(* Logix 5000 project; controller cal1632 1756-L62 rev 16.20; software revision 16.05; part 7 of 57 *)
(* tags used below, declared in another part *)
   FAULT : BOOL;
   p01_ai_prs : REAL;
   p01_ai_tc : REAL;
   p01_dint_to_hmi : DINT[16];
   p01_int_from_oxidizer : INT[10];
   p01_int_to_oxidizer : INT;
   p01_recipe_active : recipe;
   p01r03_oxidizer_prs : SYS_SCP;
   p01r03_prs_input_max : REAL;
   p01r03_prs_input_min : REAL;
   p01r03_prs_output_max : REAL;
   p01r03_prs_output_min : REAL;
   p01r09_pb_global_reset : BOOL;
   p01r14 : routine;
   p01r14_msg_read : MESSAGE;
   p01r14_msg_read_retry_timer : TIMER;
   p01r14_msg_read_timer : TIMER;
   p01r14_msg_write : MESSAGE;
   p01r14_msg_write_retry_timer : TIMER;
   p01r14_msg_write_timer : TIMER;
   p01r14_oxidizer_heart_beat_off : TIMER;
   p01r14_oxidizer_heart_beat_ok : BOOL;
   p01r14_oxidizer_heart_beat_on : TIMER;
   p01r14_oxidizer_mass_flow : REAL;
   p01r14_timer_fault : TIMER[10];
   p01r14_timer_warning : TIMER[5];
   p02_dint_from_hmi : hmi_dint;
   p02_dint_to_hmi : hmi_dint;
   p02_recipe_from_hmi : recipe;
   p02_recipe_to_hmi : recipe;
   p02r01 : routine;
   p02r02 : routine;
   p02r02_timer_fault : TIMER[4];
   p02r02_timer_logout : TIMER;
   p02r02_timer_warning : TIMER[4];
   p02r03 : routine;
   p02r03_timer_fault : TIMER[4];
   p02r03_timer_warning : TIMER[4];
   p02r04 : routine;
   p02r04_timer_fault : TIMER[4];
   p02r04_timer_warning : TIMER[4];
   p02r05 : routine;
   p02r05_timer_fault : TIMER[4];
   p02r05_timer_warning : TIMER[4];
   p02r07 : routine;
   p11_dint_to_hmi : DINT[16];
   p11r02_shutdown_temp : BOOL;
   p11r20_state : DINT;
   p11r30_request_heat : BOOL;
   p12_dint_to_hmi : DINT[16];
   p12r02_shutdown_temp : BOOL;
   p12r20_state : DINT;
   p12r30_request_heat : BOOL;
   p13_dint_to_hmi : DINT[16];
   p13r02_shutdown_temp : BOOL;
   p13r20_state : DINT;
   p13r30_request_cool : BOOL;
   p19_dint_to_hmi : DINT[16];
   p20_dint_to_hmi : DINT[16];
   p21_dint_to_hmi : DINT[16];
   p22_dint_to_hmi : DINT[16];
   p23_dint_to_hmi : DINT[32];
   p24_dint_to_hmi : DINT[16];
   p25_dint_to_hmi : DINT[16];
   p26_dint_to_hmi : DINT[16];
   p27_dint_to_hmi : DINT[16];
   p28_dint_to_hmi : DINT[16];
   p29_dint_to_hmi : DINT[16];
   p30_dint_to_hmi : DINT[16];
(* P01_System, continued *)

ROUTINE R14_Oxidizer   (* ladder *)
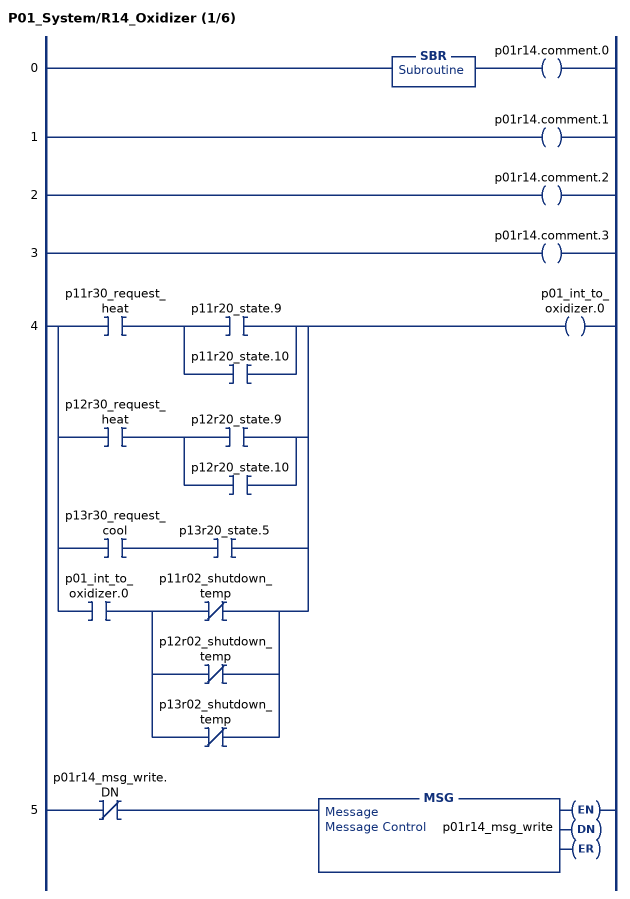
   0: SBR()OTE(p01r14.comment.0);
   1: OTE(p01r14.comment.1);
   2: OTE(p01r14.comment.2);
   3: OTE(p01r14.comment.3);
   4: [XIC(p11r30_request_heat) [XIC(p11r20_state.9) ,XIC(p11r20_state.10) ] ,XIC(p12r30_request_heat) [XIC(p12r20_state.9) ,XIC(p12r20_state.10) ] ,XIC(p13r30_request_cool) XIC(p13r20_state.5) ,XIC(p01_int_to_oxidizer.0) [XIO(p11r02_shutdown_temp) ,XIO(p12r02_shutdown_temp) ,XIO(p13r02_shutdown_temp) ] ]OTE(p01_int_to_oxidizer.0);
   5: XIO(p01r14_msg_write.DN)MSG(p01r14_msg_write);
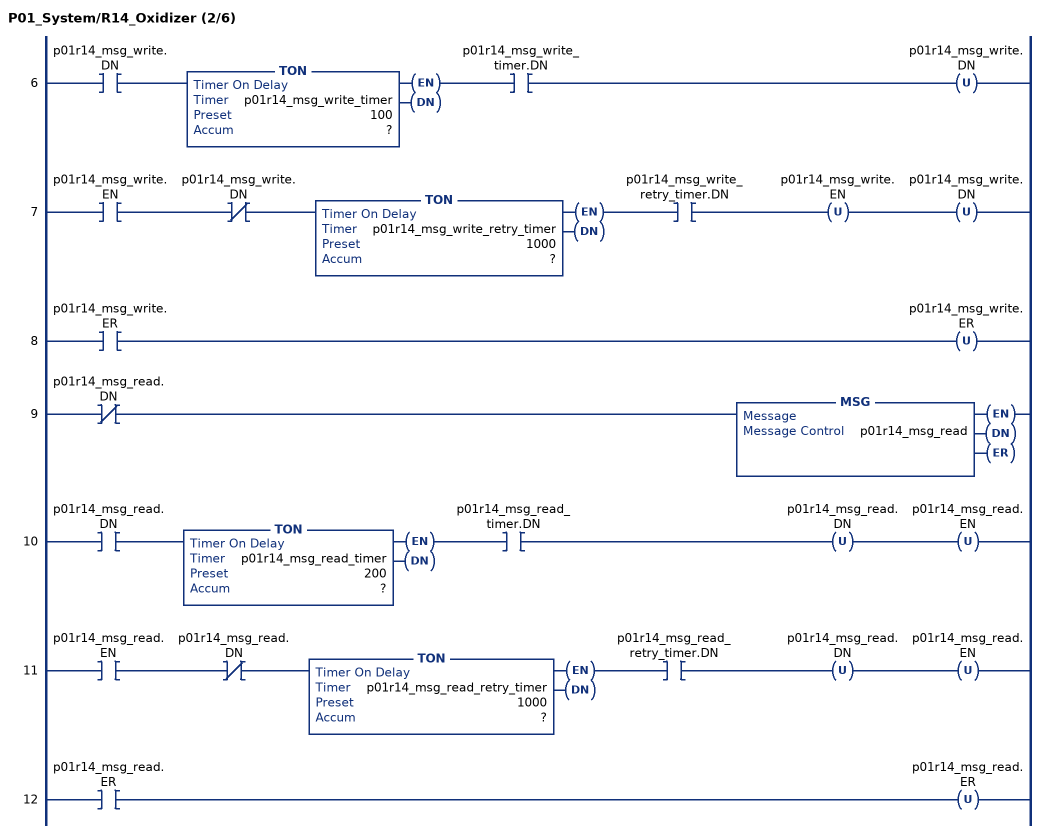
   6: XIC(p01r14_msg_write.DN)TON(p01r14_msg_write_timer,?,?)XIC(p01r14_msg_write_timer.DN)OTU(p01r14_msg_write.DN);
   7: XIC(p01r14_msg_write.EN)XIO(p01r14_msg_write.DN)TON(p01r14_msg_write_retry_timer,?,?)XIC(p01r14_msg_write_retry_timer.DN)OTU(p01r14_msg_write.EN)OTU(p01r14_msg_write.DN);
   8: XIC(p01r14_msg_write.ER)OTU(p01r14_msg_write.ER);
   9: XIO(p01r14_msg_read.DN)MSG(p01r14_msg_read);
   10: XIC(p01r14_msg_read.DN)TON(p01r14_msg_read_timer,?,?)XIC(p01r14_msg_read_timer.DN)OTU(p01r14_msg_read.DN)OTU(p01r14_msg_read.EN);
   11: XIC(p01r14_msg_read.EN)XIO(p01r14_msg_read.DN)TON(p01r14_msg_read_retry_timer,?,?)XIC(p01r14_msg_read_retry_timer.DN)OTU(p01r14_msg_read.DN)OTU(p01r14_msg_read.EN);
   12: XIC(p01r14_msg_read.ER)OTU(p01r14_msg_read.ER);
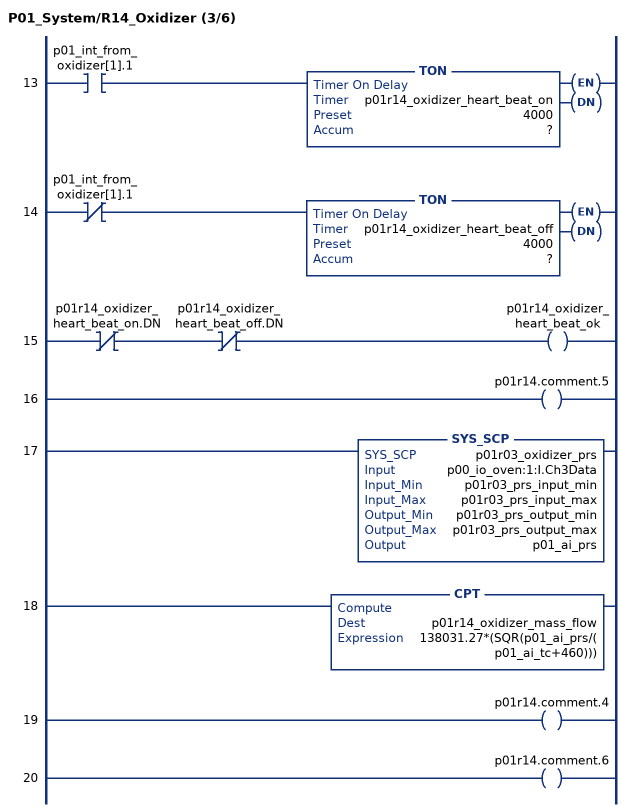
   13: XIC(p01_int_from_oxidizer[1].1)TON(p01r14_oxidizer_heart_beat_on,?,?);
   14: XIO(p01_int_from_oxidizer[1].1)TON(p01r14_oxidizer_heart_beat_off,?,?);
   15: XIO(p01r14_oxidizer_heart_beat_on.DN)XIO(p01r14_oxidizer_heart_beat_off.DN)OTE(p01r14_oxidizer_heart_beat_ok);
   16: OTE(p01r14.comment.5);
   17: SYS_SCP(p01r03_oxidizer_prs,p00_io_oven:1:I.Ch3Data,p01r03_prs_input_min,p01r03_prs_input_max,p01r03_prs_output_min,p01r03_prs_output_max,p01_ai_prs);
   18: CPT(p01r14_oxidizer_mass_flow,138031.27*(SQR(p01_ai_prs/(p01_ai_tc+460))));
   19: OTE(p01r14.comment.4);
   20: OTE(p01r14.comment.6);
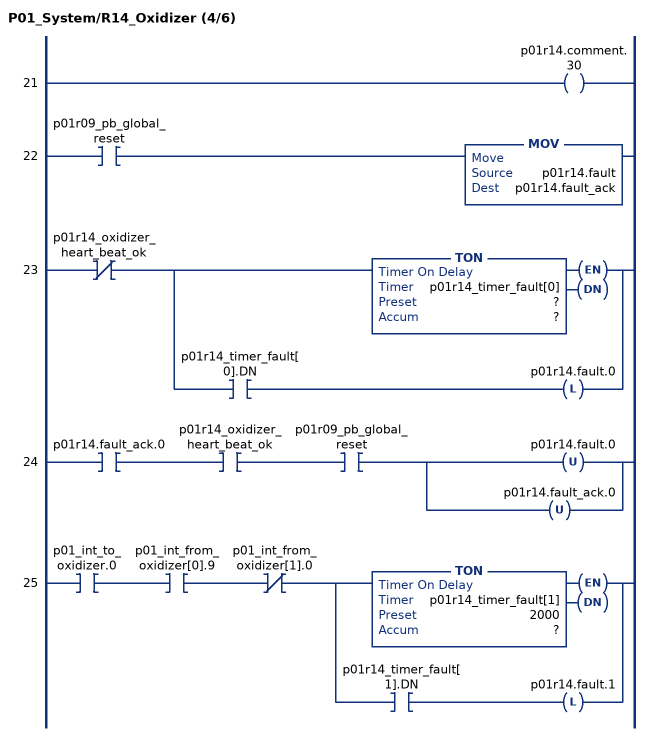
   21: OTE(p01r14.comment.30);
   22: XIC(p01r09_pb_global_reset)MOV(p01r14.fault,p01r14.fault_ack);
   23: XIO(p01r14_oxidizer_heart_beat_ok)[TON(p01r14_timer_fault[0],?,?) ,XIC(p01r14_timer_fault[0].DN) OTL(p01r14.fault.0) ];
   24: XIC(p01r14.fault_ack.0)XIC(p01r14_oxidizer_heart_beat_ok)XIC(p01r09_pb_global_reset)[OTU(p01r14.fault.0) ,OTU(p01r14.fault_ack.0) ];
   25: XIC(p01_int_to_oxidizer.0)XIC(p01_int_from_oxidizer[0].9)XIO(p01_int_from_oxidizer[1].0)[TON(p01r14_timer_fault[1],?,?) ,XIC(p01r14_timer_fault[1].DN) OTL(p01r14.fault.1) ];
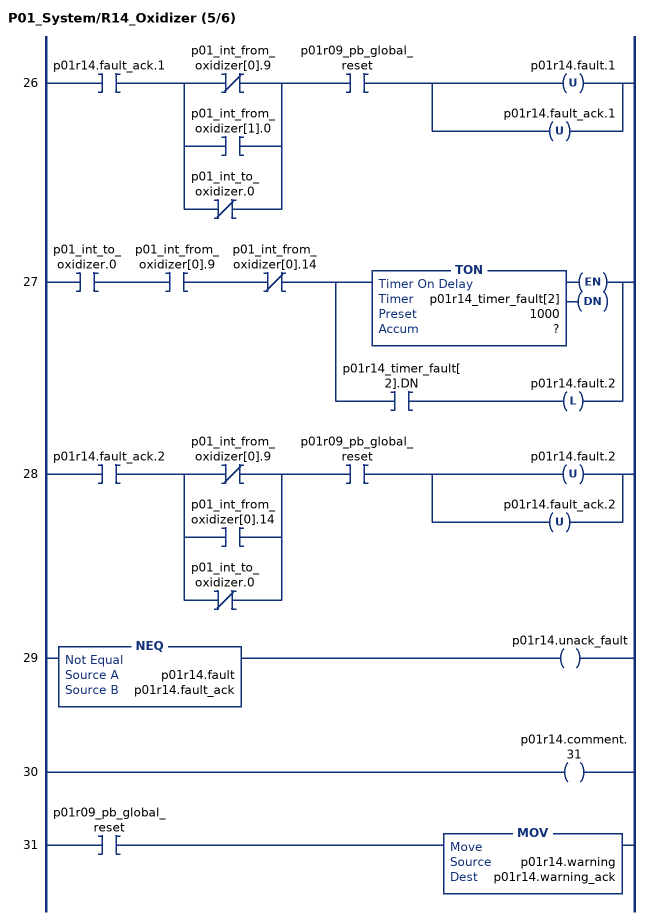
   26: XIC(p01r14.fault_ack.1)[XIO(p01_int_from_oxidizer[0].9) ,XIC(p01_int_from_oxidizer[1].0) ,XIO(p01_int_to_oxidizer.0) ]XIC(p01r09_pb_global_reset)[OTU(p01r14.fault.1) ,OTU(p01r14.fault_ack.1) ];
   27: XIC(p01_int_to_oxidizer.0)XIC(p01_int_from_oxidizer[0].9)XIO(p01_int_from_oxidizer[0].14)[TON(p01r14_timer_fault[2],?,?) ,XIC(p01r14_timer_fault[2].DN) OTL(p01r14.fault.2) ];
   28: XIC(p01r14.fault_ack.2)[XIO(p01_int_from_oxidizer[0].9) ,XIC(p01_int_from_oxidizer[0].14) ,XIO(p01_int_to_oxidizer.0) ]XIC(p01r09_pb_global_reset)[OTU(p01r14.fault.2) ,OTU(p01r14.fault_ack.2) ];
   29: NEQ(p01r14.fault,p01r14.fault_ack)OTE(p01r14.unack_fault);
   30: OTE(p01r14.comment.31);
   31: XIC(p01r09_pb_global_reset)MOV(p01r14.warning,p01r14.warning_ack);
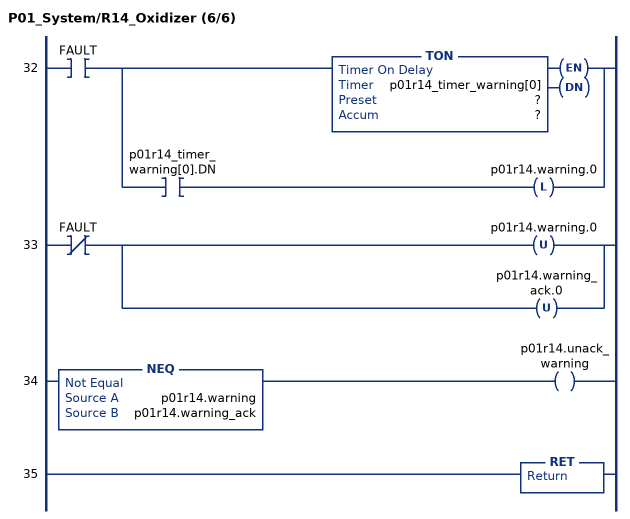
   32: XIC(FAULT)[TON(p01r14_timer_warning[0],?,?) ,XIC(p01r14_timer_warning[0].DN) OTL(p01r14.warning.0) ];
   33: XIO(FAULT)[OTU(p01r14.warning.0) ,OTU(p01r14.warning_ack.0) ];
   34: NEQ(p01r14.warning,p01r14.warning_ack)OTE(p01r14.unack_warning);
   35: RET();
END_ROUTINE
END_PROGRAM

PROGRAM P02_MOP_HMI_Iface   (* main routine R01_Main *)

ROUTINE R01_Main   (* ladder *)
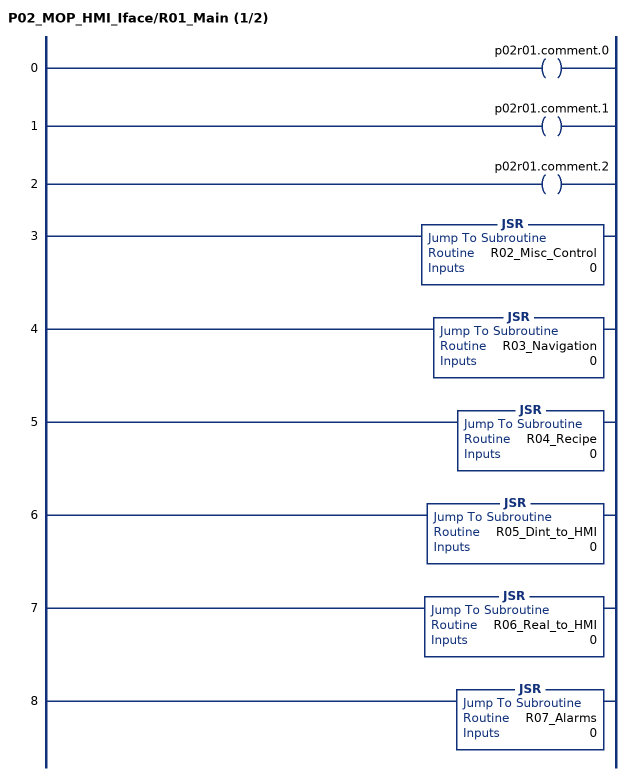
   0: OTE(p02r01.comment.0);
   1: OTE(p02r01.comment.1);
   2: OTE(p02r01.comment.2);
   3: JSR(R02_Misc_Control,0);
   4: JSR(R03_Navigation,0);
   5: JSR(R04_Recipe,0);
   6: JSR(R05_Dint_to_HMI,0);
   7: JSR(R06_Real_to_HMI,0);
   8: JSR(R07_Alarms,0);
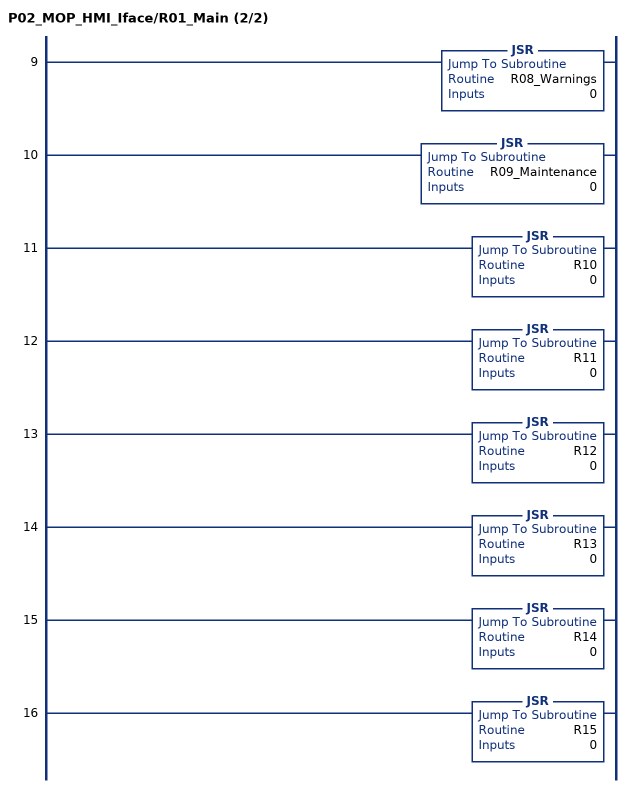
   9: JSR(R08_Warnings,0);
   10: JSR(R09_Maintenance,0);
   11: JSR(R10,0);
   12: JSR(R11,0);
   13: JSR(R12,0);
   14: JSR(R13,0);
   15: JSR(R14,0);
   16: JSR(R15,0);
END_ROUTINE

ROUTINE R02_Misc_Control   (* ladder *)
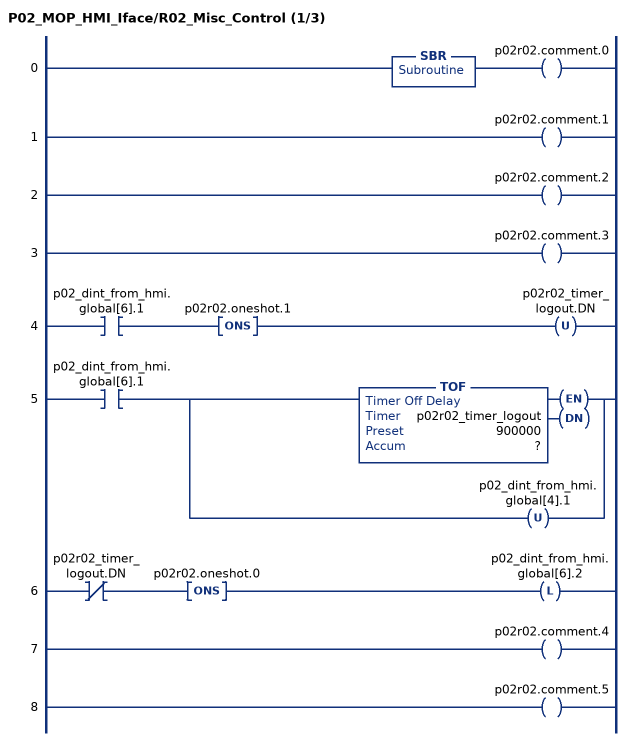
   0: SBR()OTE(p02r02.comment.0);
   1: OTE(p02r02.comment.1);
   2: OTE(p02r02.comment.2);
   3: OTE(p02r02.comment.3);
   4: XIC(p02_dint_from_hmi.global[6].1)ONS(p02r02.oneshot.1)OTU(p02r02_timer_logout.DN);
   5: XIC(p02_dint_from_hmi.global[6].1)[TOF(p02r02_timer_logout,?,?) ,OTU(p02_dint_from_hmi.global[4].1) ];
   6: XIO(p02r02_timer_logout.DN)ONS(p02r02.oneshot.0)OTL(p02_dint_from_hmi.global[6].2);
   7: OTE(p02r02.comment.4);
   8: OTE(p02r02.comment.5);
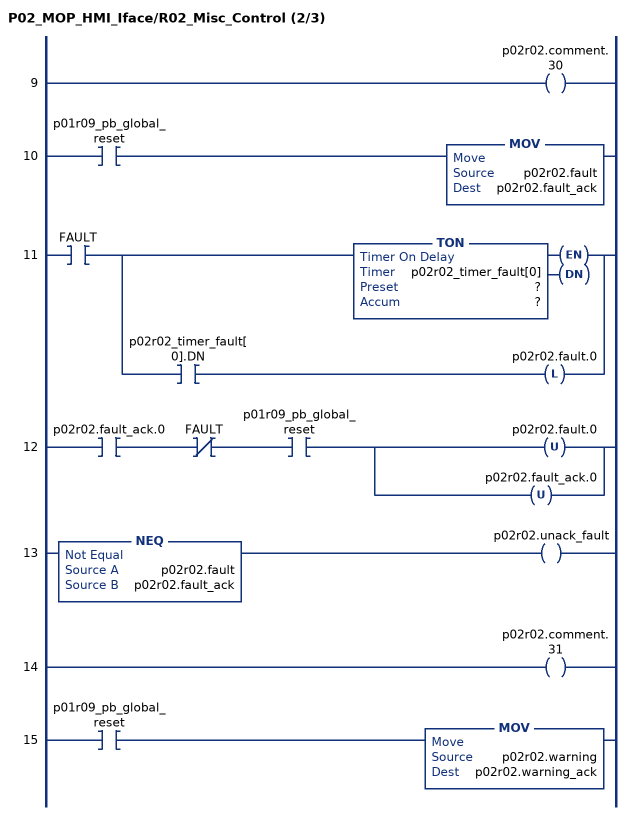
   9: OTE(p02r02.comment.30);
   10: XIC(p01r09_pb_global_reset)MOV(p02r02.fault,p02r02.fault_ack);
   11: XIC(FAULT)[TON(p02r02_timer_fault[0],?,?) ,XIC(p02r02_timer_fault[0].DN) OTL(p02r02.fault.0) ];
   12: XIC(p02r02.fault_ack.0)XIO(FAULT)XIC(p01r09_pb_global_reset)[OTU(p02r02.fault.0) ,OTU(p02r02.fault_ack.0) ];
   13: NEQ(p02r02.fault,p02r02.fault_ack)OTE(p02r02.unack_fault);
   14: OTE(p02r02.comment.31);
   15: XIC(p01r09_pb_global_reset)MOV(p02r02.warning,p02r02.warning_ack);
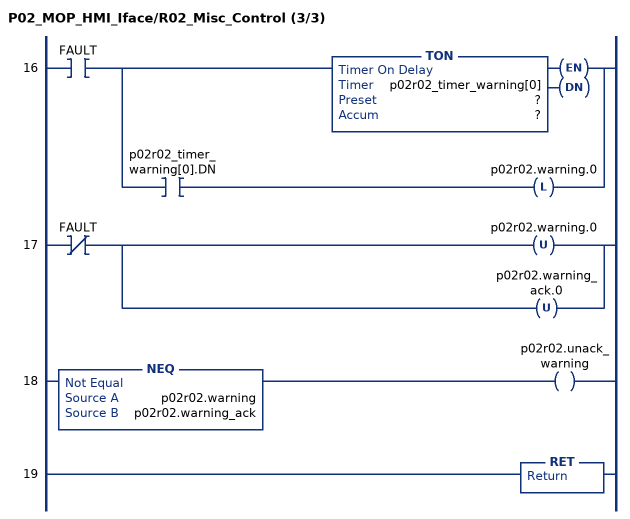
   16: XIC(FAULT)[TON(p02r02_timer_warning[0],?,?) ,XIC(p02r02_timer_warning[0].DN) OTL(p02r02.warning.0) ];
   17: XIO(FAULT)[OTU(p02r02.warning.0) ,OTU(p02r02.warning_ack.0) ];
   18: NEQ(p02r02.warning,p02r02.warning_ack)OTE(p02r02.unack_warning);
   19: RET();
END_ROUTINE

ROUTINE R03_Navigation   (* ladder *)
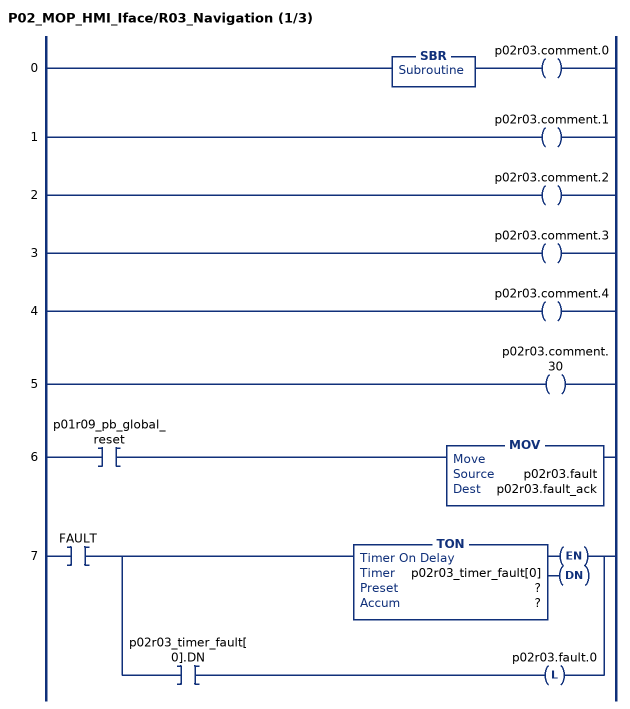
   0: SBR()OTE(p02r03.comment.0);
   1: OTE(p02r03.comment.1);
   2: OTE(p02r03.comment.2);
   3: OTE(p02r03.comment.3);
   4: OTE(p02r03.comment.4);
   5: OTE(p02r03.comment.30);
   6: XIC(p01r09_pb_global_reset)MOV(p02r03.fault,p02r03.fault_ack);
   7: XIC(FAULT)[TON(p02r03_timer_fault[0],?,?) ,XIC(p02r03_timer_fault[0].DN) OTL(p02r03.fault.0) ];
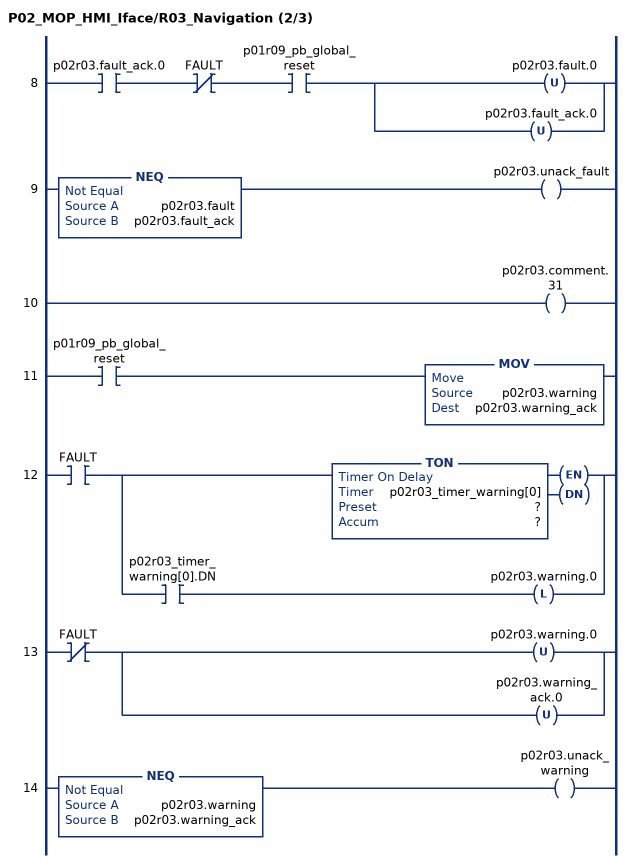
   8: XIC(p02r03.fault_ack.0)XIO(FAULT)XIC(p01r09_pb_global_reset)[OTU(p02r03.fault.0) ,OTU(p02r03.fault_ack.0) ];
   9: NEQ(p02r03.fault,p02r03.fault_ack)OTE(p02r03.unack_fault);
   10: OTE(p02r03.comment.31);
   11: XIC(p01r09_pb_global_reset)MOV(p02r03.warning,p02r03.warning_ack);
   12: XIC(FAULT)[TON(p02r03_timer_warning[0],?,?) ,XIC(p02r03_timer_warning[0].DN) OTL(p02r03.warning.0) ];
   13: XIO(FAULT)[OTU(p02r03.warning.0) ,OTU(p02r03.warning_ack.0) ];
   14: NEQ(p02r03.warning,p02r03.warning_ack)OTE(p02r03.unack_warning);
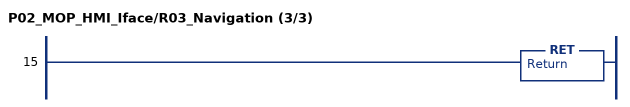
   15: RET();
END_ROUTINE

ROUTINE R04_Recipe   (* ladder *)
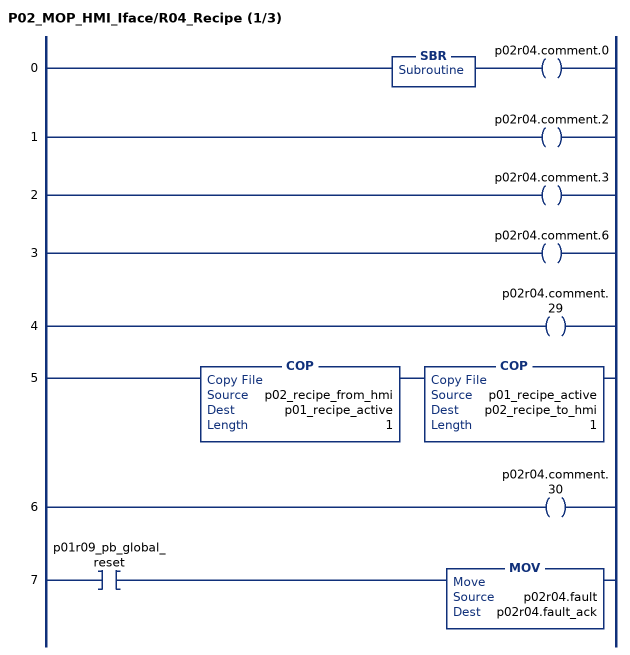
   0: SBR()OTE(p02r04.comment.0);
   1: OTE(p02r04.comment.2);
   2: OTE(p02r04.comment.3);
   3: OTE(p02r04.comment.6);
   4: OTE(p02r04.comment.29);
   5: COP(p02_recipe_from_hmi,p01_recipe_active,1)COP(p01_recipe_active,p02_recipe_to_hmi,1);
   6: OTE(p02r04.comment.30);
   7: XIC(p01r09_pb_global_reset)MOV(p02r04.fault,p02r04.fault_ack);
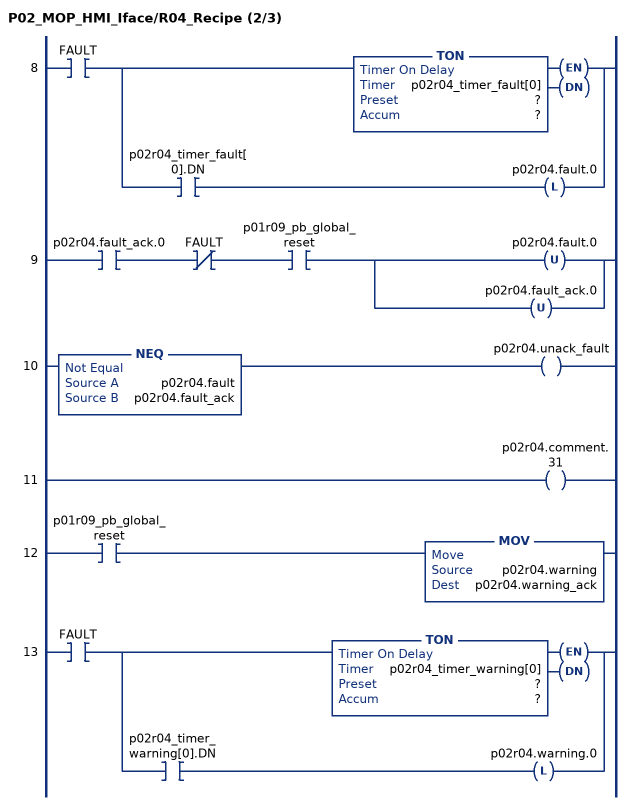
   8: XIC(FAULT)[TON(p02r04_timer_fault[0],?,?) ,XIC(p02r04_timer_fault[0].DN) OTL(p02r04.fault.0) ];
   9: XIC(p02r04.fault_ack.0)XIO(FAULT)XIC(p01r09_pb_global_reset)[OTU(p02r04.fault.0) ,OTU(p02r04.fault_ack.0) ];
   10: NEQ(p02r04.fault,p02r04.fault_ack)OTE(p02r04.unack_fault);
   11: OTE(p02r04.comment.31);
   12: XIC(p01r09_pb_global_reset)MOV(p02r04.warning,p02r04.warning_ack);
   13: XIC(FAULT)[TON(p02r04_timer_warning[0],?,?) ,XIC(p02r04_timer_warning[0].DN) OTL(p02r04.warning.0) ];
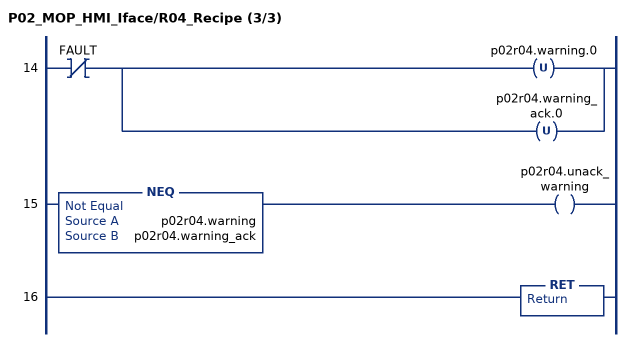
   14: XIO(FAULT)[OTU(p02r04.warning.0) ,OTU(p02r04.warning_ack.0) ];
   15: NEQ(p02r04.warning,p02r04.warning_ack)OTE(p02r04.unack_warning);
   16: RET();
END_ROUTINE

ROUTINE R05_Dint_to_HMI   (* ladder *)
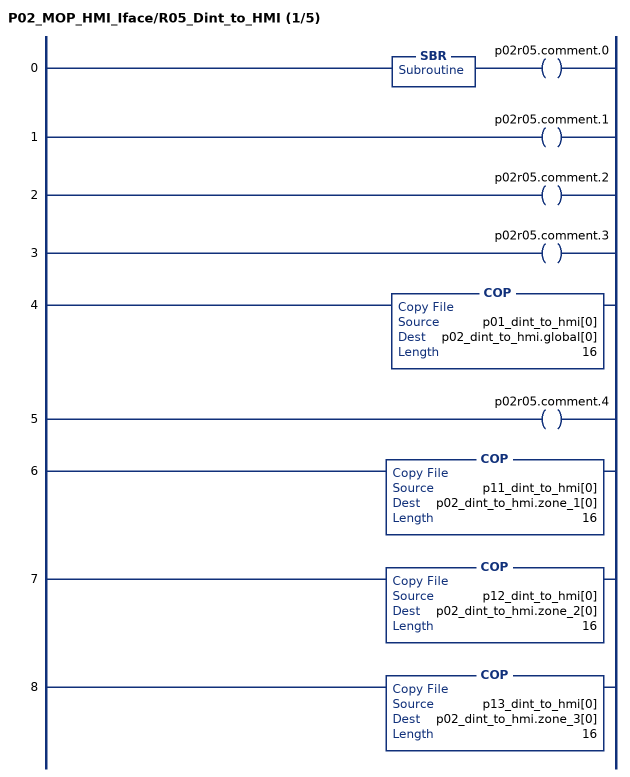
   0: SBR()OTE(p02r05.comment.0);
   1: OTE(p02r05.comment.1);
   2: OTE(p02r05.comment.2);
   3: OTE(p02r05.comment.3);
   4: COP(p01_dint_to_hmi[0],p02_dint_to_hmi.global[0],16);
   5: OTE(p02r05.comment.4);
   6: COP(p11_dint_to_hmi[0],p02_dint_to_hmi.zone_1[0],16);
   7: COP(p12_dint_to_hmi[0],p02_dint_to_hmi.zone_2[0],16);
   8: COP(p13_dint_to_hmi[0],p02_dint_to_hmi.zone_3[0],16);
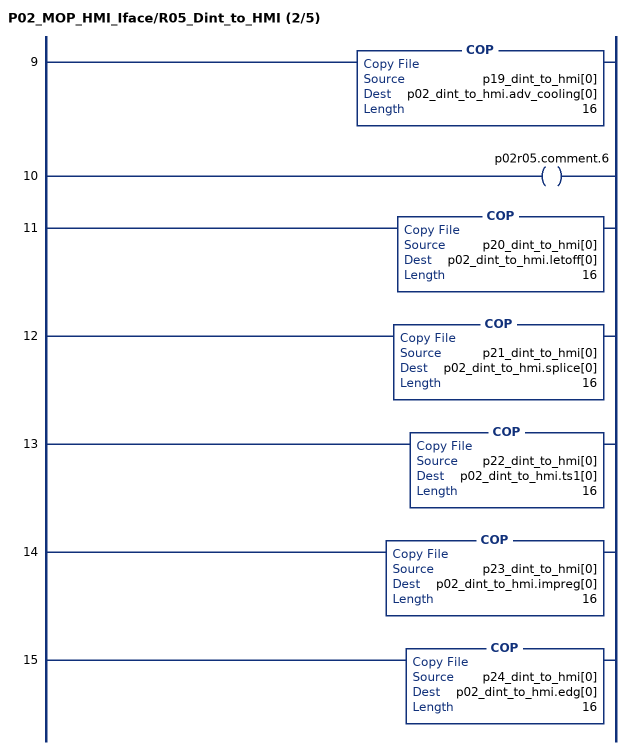
   9: COP(p19_dint_to_hmi[0],p02_dint_to_hmi.adv_cooling[0],16);
   10: OTE(p02r05.comment.6);
   11: COP(p20_dint_to_hmi[0],p02_dint_to_hmi.letoff[0],16);
   12: COP(p21_dint_to_hmi[0],p02_dint_to_hmi.splice[0],16);
   13: COP(p22_dint_to_hmi[0],p02_dint_to_hmi.ts1[0],16);
   14: COP(p23_dint_to_hmi[0],p02_dint_to_hmi.impreg[0],16);
   15: COP(p24_dint_to_hmi[0],p02_dint_to_hmi.edg[0],16);
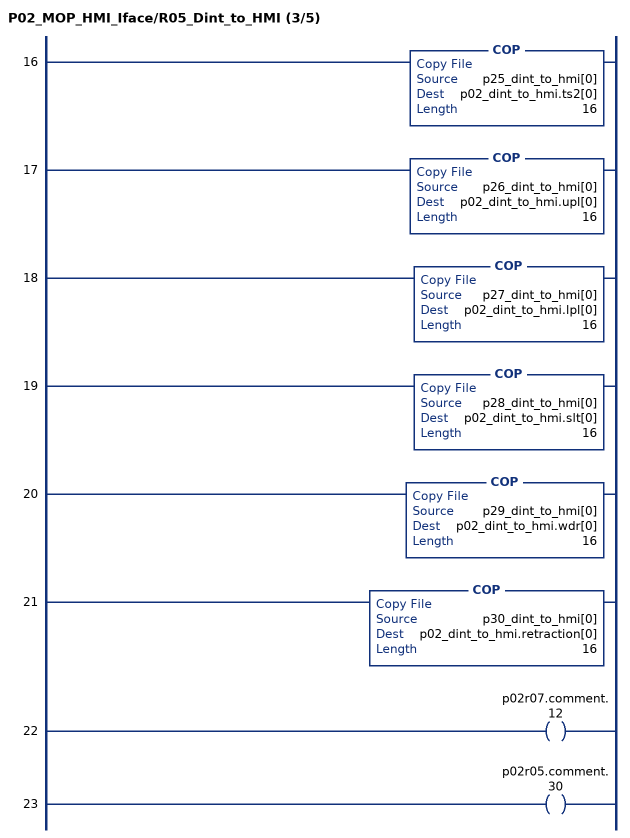
   16: COP(p25_dint_to_hmi[0],p02_dint_to_hmi.ts2[0],16);
   17: COP(p26_dint_to_hmi[0],p02_dint_to_hmi.upl[0],16);
   18: COP(p27_dint_to_hmi[0],p02_dint_to_hmi.lpl[0],16);
   19: COP(p28_dint_to_hmi[0],p02_dint_to_hmi.slt[0],16);
   20: COP(p29_dint_to_hmi[0],p02_dint_to_hmi.wdr[0],16);
   21: COP(p30_dint_to_hmi[0],p02_dint_to_hmi.retraction[0],16);
   22: OTE(p02r07.comment.12);
   23: OTE(p02r05.comment.30);
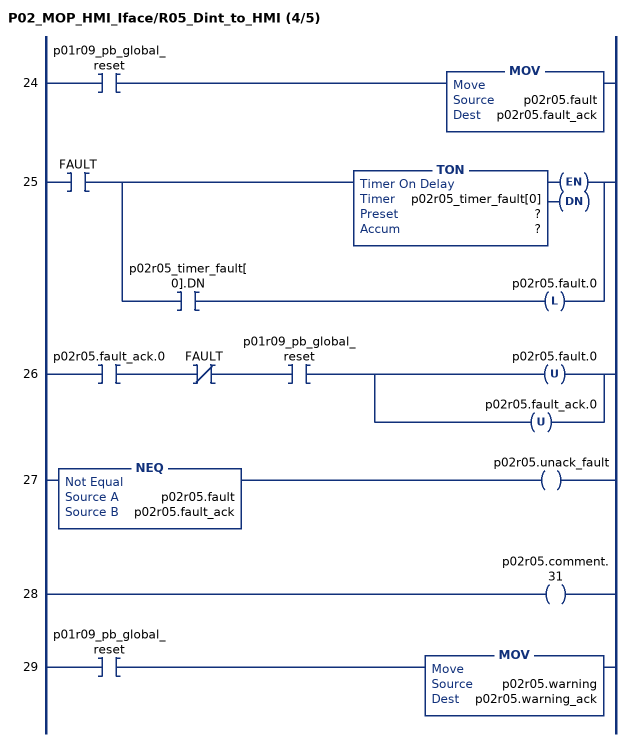
   24: XIC(p01r09_pb_global_reset)MOV(p02r05.fault,p02r05.fault_ack);
   25: XIC(FAULT)[TON(p02r05_timer_fault[0],?,?) ,XIC(p02r05_timer_fault[0].DN) OTL(p02r05.fault.0) ];
   26: XIC(p02r05.fault_ack.0)XIO(FAULT)XIC(p01r09_pb_global_reset)[OTU(p02r05.fault.0) ,OTU(p02r05.fault_ack.0) ];
   27: NEQ(p02r05.fault,p02r05.fault_ack)OTE(p02r05.unack_fault);
   28: OTE(p02r05.comment.31);
   29: XIC(p01r09_pb_global_reset)MOV(p02r05.warning,p02r05.warning_ack);
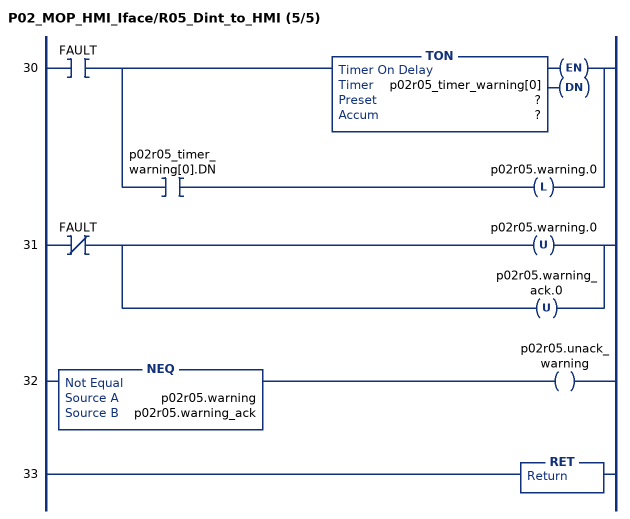
   30: XIC(FAULT)[TON(p02r05_timer_warning[0],?,?) ,XIC(p02r05_timer_warning[0].DN) OTL(p02r05.warning.0) ];
   31: XIO(FAULT)[OTU(p02r05.warning.0) ,OTU(p02r05.warning_ack.0) ];
   32: NEQ(p02r05.warning,p02r05.warning_ack)OTE(p02r05.unack_warning);
   33: RET();
END_ROUTINE
